// TIA Portal V19 export
DATA_BLOCK "DB_Alarme"   // DB1201
{ S7_Optimized_Access := 'TRUE' }
// stored: AutoNumber false, MemoryReserve 100
   VAR RETAIN
      MLD : Array[0.."Anzahl_Alarm_Woerter"] of Word;
      AM_MLD : Array[0.."Anzahl_Alarm_Woerter"] of Word;
      Para_Mld : Array[0.."Anzahl_Alarm_Woerter"] of "Alarm_Parameter_Wort";   // Struct = Meldewort, Array = ParaByte für MeldeBit (siehe FC5)
      WrnM : Array[0..1] of Word;
      Edit : Struct
         Edit_Meld : Int := 1;   // aktuell zu editierende Meldung
         Edit_Meld_old : Int;
         Edit_Meldewort : Int;   // betroffenes Meldewort
         Edit_Meldebit : Int;   // betroffenes Meldebit
         AM_Edit : Bool;
         Uebernehmen : Bool;   // Änderungen Übernehmen
         Uebernommen : Bool;   // Änderungen für ausgewählte Meldung übernommen
         Verwerfen : Bool;   // Änderungen verwerfen
         Editiert : Bool;   // Alarm wurde geändert
         Par : "Alarm_Parameter";
      END_STRUCT;
      auto_aus : Bool;
      stop_request : Bool;
      Sammelbit_St : Bool;
      Sammelbit_Wrn : Bool;
      M_Q_Hupe_Rot : Bool;
      M_Q_Hupe_Gelb : Bool;
      M_Q_Hupe_Blau : Bool;
      Hupe_Dauer_Rot : Bool;
      Hupe_Dauer_Gelb : Bool;
      Hupe_Dauer_Blau : Bool;
      IN_Quitt_Hupe : Bool;
      AM_T_Hupe : Bool;
      La_Quit_Err : Bool;   // Lampe Fehlerquittung
      Lampe_Rot : Bool;
      Lampe_Gelb : Bool;
      Lampe_Blau : Bool;
      Zeit_Auto_Quitt_Hupe_Rot : Time_Of_Day := TOD#00:00:05;
      Zeit_Auto_Quitt_Hupe_Gelb : Time_Of_Day := TOD#00:00:05;
      Zeit_Auto_Quitt_Hupe_Blau : Time_Of_Day := TOD#00:00:05;
      Timer_Hupe_Rot : TON_TIME;
      Timer_Hupe_Gelb : TON_TIME;
      Timer_Hupe_Blau : TON_TIME;
   END_VAR
BEGIN
END_DATA_BLOCK
